// Mitsubishi GX Works2 project: Jesús Beato 2023-1283 #5   PLC: FX2N/FX2NC

PROGRAM MAIN
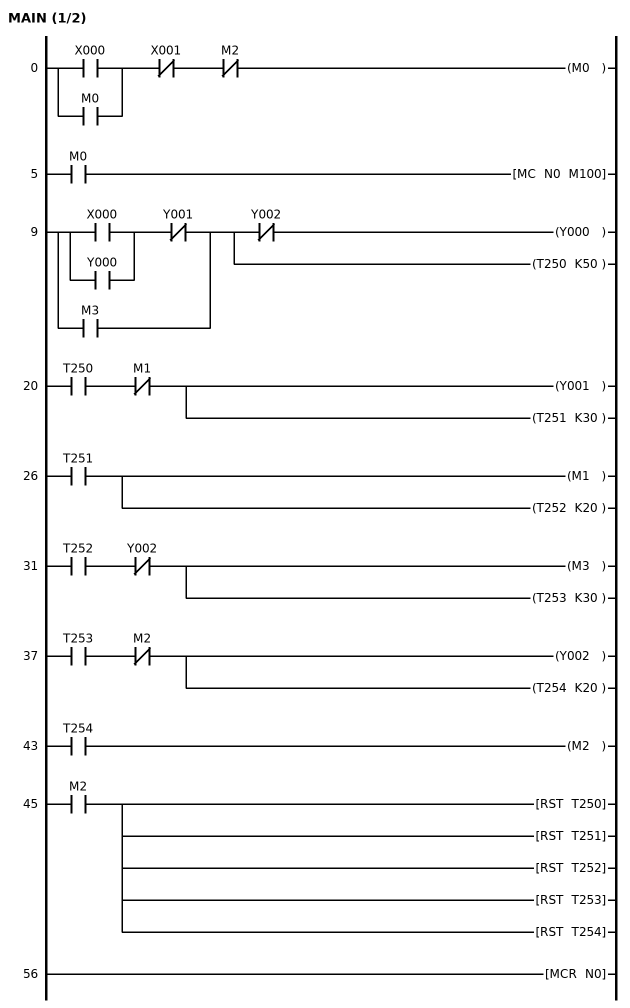
0     LD      X000
      OR      M0
      ANI     X001
      ANI     M2
      OUT     M0
5     LD      M0
      MC      N0 M100
9     LD      X000
      OR      Y000
      ANI     Y001
      OR      M3
      MPS
      ANI     Y002
      OUT     Y000
      MPP
      OUT     T250 K50
20    LD      T250
      ANI     M1
      OUT     Y001
      OUT     T251 K30
26    LD      T251
      OUT     M1
      OUT     T252 K20
31    LD      T252
      ANI     Y002
      OUT     M3
      OUT     T253 K30
37    LD      T253
      ANI     M2
      OUT     Y002
      OUT     T254 K20
43    LD      T254
      OUT     M2
45    LD      M2
      RST     T250
      RST     T251
      RST     T252
      RST     T253
      RST     T254
56    MCR     N0
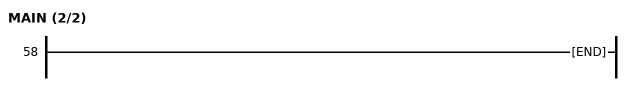
58    END
END_PROGRAM
